PROGRAM MAIN
VAR
END_VAR

END_PROGRAM

(* stored: Version 1.1.0.1
   POU MAIN: Id {b5059249-4135-4e8e-8f8f-20897623daea} *)
